FUNCTION F_Any_To_Generic : T_Generic
VAR_INPUT
	Value : ANY;
END_VAR

F_Any_To_Generic := Value;

END_FUNCTION

(* stored: Version 1.1.0.1, ProductVersion 3.1.4024.4
   POU F_Any_To_Generic: Id {4ace65b1-964e-4cd2-9d38-592d2c551f06}, SpecialFunc None *)
